Staubli VAL3: checkTollerance.pgx

public program checkTollerance(bool& x_bOk (dimensions=1))
begin
  if distance(here(flange,world),pTollerance)<nTollerance
    x_bOk=true
  else
    x_bOk=false
  endIf
end
